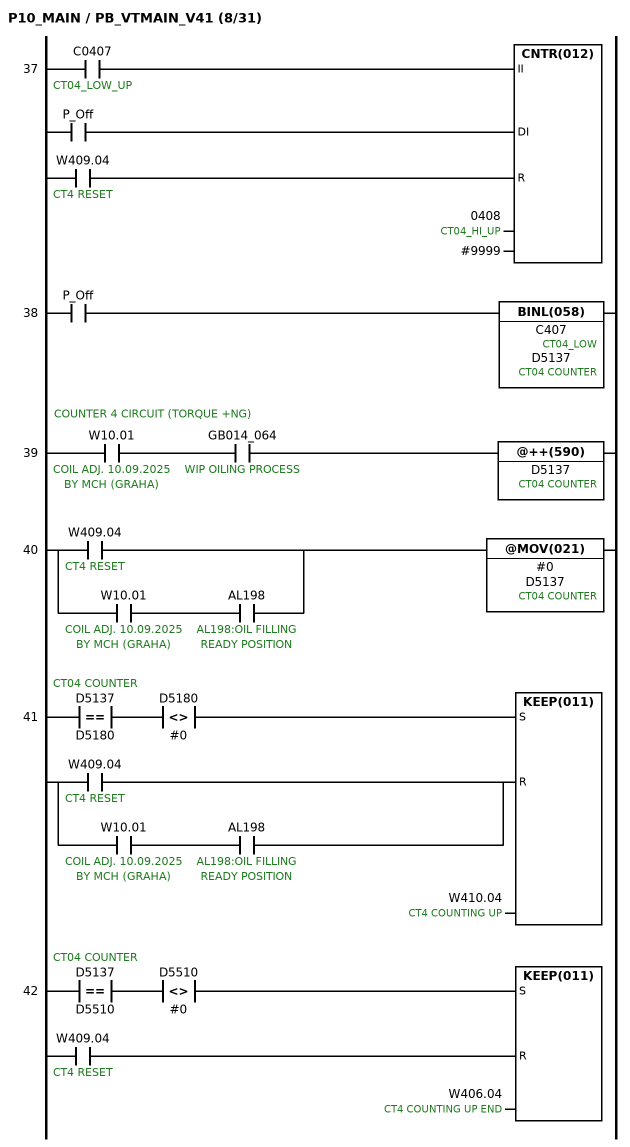
; [picture p96: P10_MAIN / PB_VTMAIN_V41, rungs 37-42]
; rung 37
LD C0407  ; CT04_LOW_UP
LD P_Off
LD W409.04  ; CT4 RESET
CNTR(012) 0408 #9999  ; CT04_HI_UP
; rung 38
LD P_Off
BINL(058) C407 D5137  ; CT04_LOW, CT04 COUNTER
; rung 39: COUNTER 4 CIRCUIT (TORQUE +NG)
LD W10.01  ; COIL ADJ. 10.09.2025 BY MCH (GRAHA)
AND GB014_064  ; WIP OILING PROCESS
@++(590) D5137  ; CT04 COUNTER
; rung 40
LD W409.04  ; CT4 RESET
LD W10.01  ; COIL ADJ. 10.09.2025 BY MCH (GRAHA)
AND AL198  ; AL198:OIL FILLING READY POSITION
ORLD
@MOV(021) #0 D5137  ; CT04 COUNTER
; rung 41
LD=L(301) D5137 D5180  ; CT04 COUNTER
AND<>L(306) D5180 #0
LD W409.04  ; CT4 RESET
LD W10.01  ; COIL ADJ. 10.09.2025 BY MCH (GRAHA)
AND AL198  ; AL198:OIL FILLING READY POSITION
ORLD
KEEP(011) W410.04  ; CT4 COUNTING UP
; rung 42
LD=L(301) D5137 D5510  ; CT04 COUNTER
AND<>L(306) D5510 #0
LD W409.04  ; CT4 RESET
KEEP(011) W406.04  ; CT4 COUNTING UP END

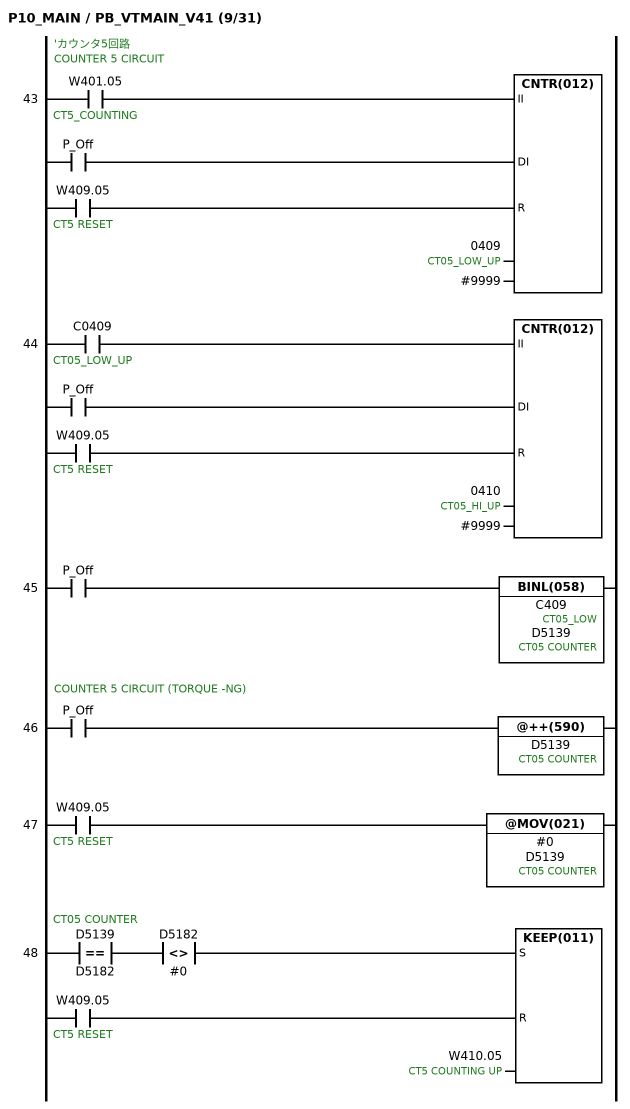
; rung 43: 'カウンタ5回路 / COUNTER 5 CIRCUIT
LD W401.05  ; CT5_COUNTING
LD P_Off
LD W409.05  ; CT5 RESET
CNTR(012) 0409 #9999  ; CT05_LOW_UP
; rung 44
LD C0409  ; CT05_LOW_UP
LD P_Off
LD W409.05  ; CT5 RESET
CNTR(012) 0410 #9999  ; CT05_HI_UP
; rung 45
LD P_Off
BINL(058) C409 D5139  ; CT05_LOW, CT05 COUNTER
; rung 46: COUNTER 5 CIRCUIT (TORQUE -NG)
LD P_Off
@++(590) D5139  ; CT05 COUNTER
; rung 47
LD W409.05  ; CT5 RESET
@MOV(021) #0 D5139  ; CT05 COUNTER
; rung 48
LD=L(301) D5139 D5182  ; CT05 COUNTER
AND<>L(306) D5182 #0
LD W409.05  ; CT5 RESET
KEEP(011) W410.05  ; CT5 COUNTING UP

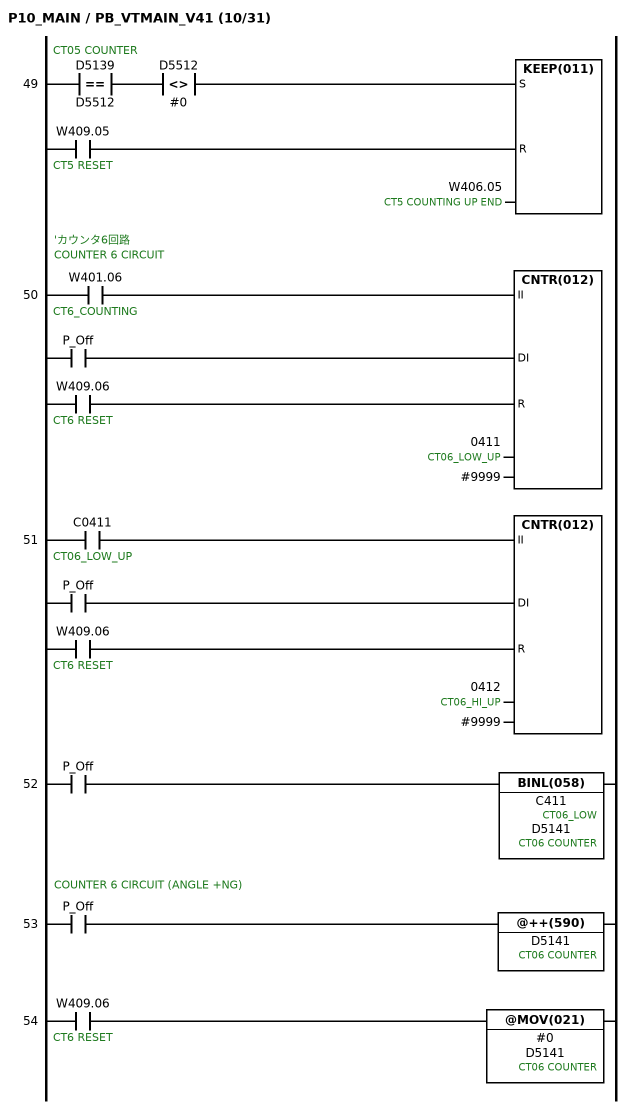
; rung 49
LD=L(301) D5139 D5512  ; CT05 COUNTER
AND<>L(306) D5512 #0
LD W409.05  ; CT5 RESET
KEEP(011) W406.05  ; CT5 COUNTING UP END
; rung 50: 'カウンタ6回路 / COUNTER 6 CIRCUIT
LD W401.06  ; CT6_COUNTING
LD P_Off
LD W409.06  ; CT6 RESET
CNTR(012) 0411 #9999  ; CT06_LOW_UP
; rung 51
LD C0411  ; CT06_LOW_UP
LD P_Off
LD W409.06  ; CT6 RESET
CNTR(012) 0412 #9999  ; CT06_HI_UP
; rung 52
LD P_Off
BINL(058) C411 D5141  ; CT06_LOW, CT06 COUNTER
; rung 53: COUNTER 6 CIRCUIT (ANGLE +NG)
LD P_Off
@++(590) D5141  ; CT06 COUNTER
; rung 54
LD W409.06  ; CT6 RESET
@MOV(021) #0 D5141  ; CT06 COUNTER

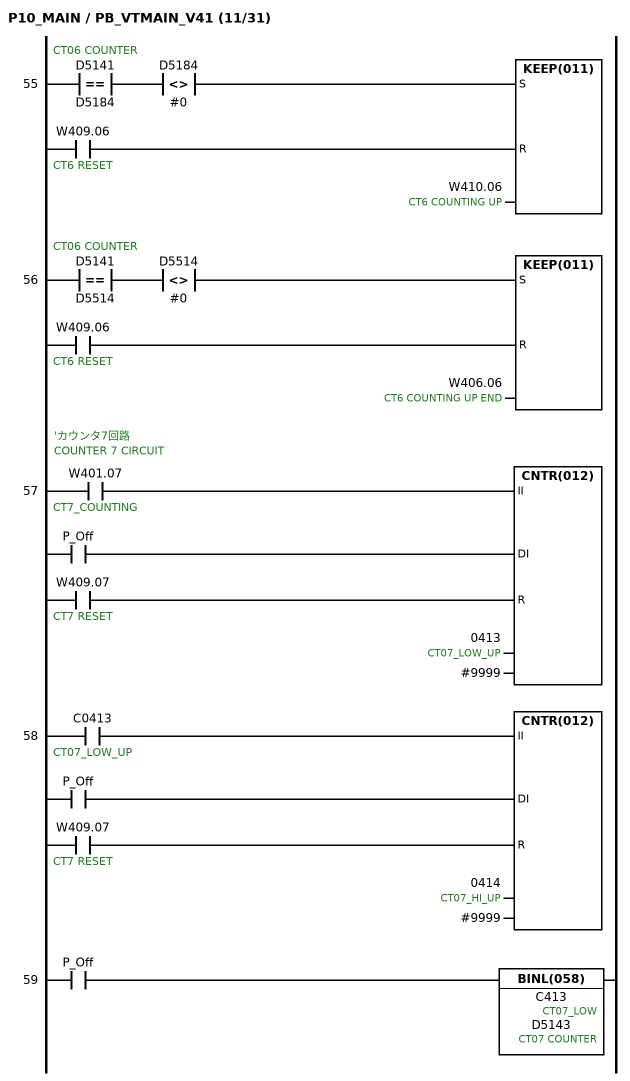
; rung 55
LD=L(301) D5141 D5184  ; CT06 COUNTER
AND<>L(306) D5184 #0
LD W409.06  ; CT6 RESET
KEEP(011) W410.06  ; CT6 COUNTING UP
; rung 56
LD=L(301) D5141 D5514  ; CT06 COUNTER
AND<>L(306) D5514 #0
LD W409.06  ; CT6 RESET
KEEP(011) W406.06  ; CT6 COUNTING UP END
; rung 57: 'カウンタ7回路 / COUNTER 7 CIRCUIT
LD W401.07  ; CT7_COUNTING
LD P_Off
LD W409.07  ; CT7 RESET
CNTR(012) 0413 #9999  ; CT07_LOW_UP
; rung 58
LD C0413  ; CT07_LOW_UP
LD P_Off
LD W409.07  ; CT7 RESET
CNTR(012) 0414 #9999  ; CT07_HI_UP
; rung 59
LD P_Off
BINL(058) C413 D5143  ; CT07_LOW, CT07 COUNTER

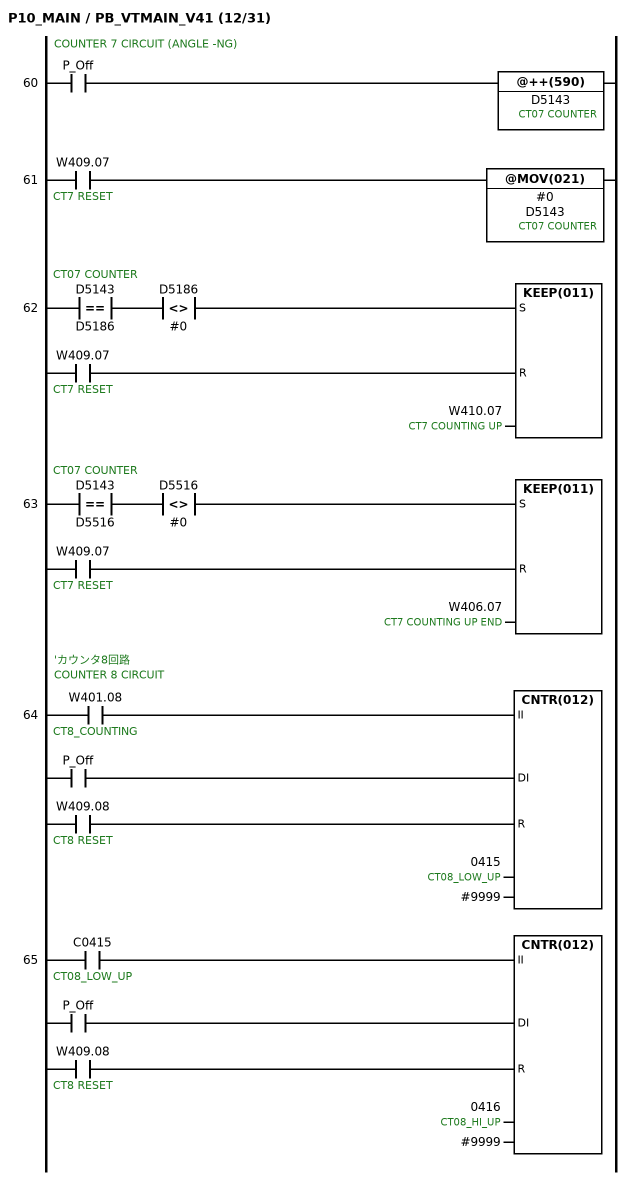
; rung 60: COUNTER 7 CIRCUIT (ANGLE -NG)
LD P_Off
@++(590) D5143  ; CT07 COUNTER
; rung 61
LD W409.07  ; CT7 RESET
@MOV(021) #0 D5143  ; CT07 COUNTER
; rung 62
LD=L(301) D5143 D5186  ; CT07 COUNTER
AND<>L(306) D5186 #0
LD W409.07  ; CT7 RESET
KEEP(011) W410.07  ; CT7 COUNTING UP
; rung 63
LD=L(301) D5143 D5516  ; CT07 COUNTER
AND<>L(306) D5516 #0
LD W409.07  ; CT7 RESET
KEEP(011) W406.07  ; CT7 COUNTING UP END
; rung 64: 'カウンタ8回路 / COUNTER 8 CIRCUIT
LD W401.08  ; CT8_COUNTING
LD P_Off
LD W409.08  ; CT8 RESET
CNTR(012) 0415 #9999  ; CT08_LOW_UP
; rung 65
LD C0415  ; CT08_LOW_UP
LD P_Off
LD W409.08  ; CT8 RESET
CNTR(012) 0416 #9999  ; CT08_HI_UP

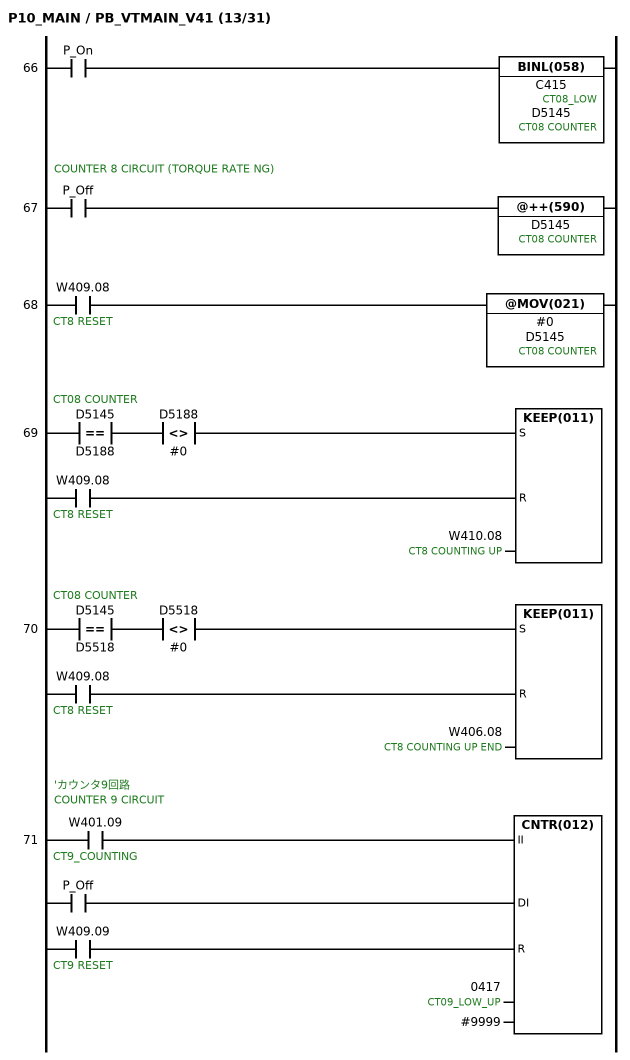
; rung 66
LD P_On
BINL(058) C415 D5145  ; CT08_LOW, CT08 COUNTER
; rung 67: COUNTER 8 CIRCUIT (TORQUE RATE NG)
LD P_Off
@++(590) D5145  ; CT08 COUNTER
; rung 68
LD W409.08  ; CT8 RESET
@MOV(021) #0 D5145  ; CT08 COUNTER
; rung 69
LD=L(301) D5145 D5188  ; CT08 COUNTER
AND<>L(306) D5188 #0
LD W409.08  ; CT8 RESET
KEEP(011) W410.08  ; CT8 COUNTING UP
; rung 70
LD=L(301) D5145 D5518  ; CT08 COUNTER
AND<>L(306) D5518 #0
LD W409.08  ; CT8 RESET
KEEP(011) W406.08  ; CT8 COUNTING UP END
; rung 71: 'カウンタ9回路 / COUNTER 9 CIRCUIT
LD W401.09  ; CT9_COUNTING
LD P_Off
LD W409.09  ; CT9 RESET
CNTR(012) 0417 #9999  ; CT09_LOW_UP

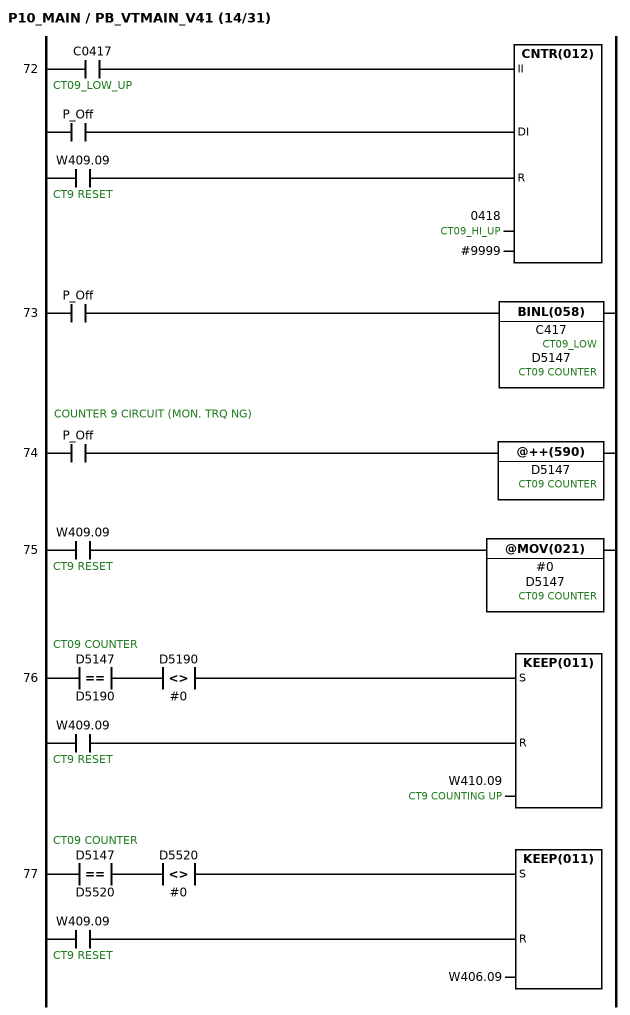
; rung 72
LD C0417  ; CT09_LOW_UP
LD P_Off
LD W409.09  ; CT9 RESET
CNTR(012) 0418 #9999  ; CT09_HI_UP
; rung 73
LD P_Off
BINL(058) C417 D5147  ; CT09_LOW, CT09 COUNTER
; rung 74: COUNTER 9 CIRCUIT (MON. TRQ NG)
LD P_Off
@++(590) D5147  ; CT09 COUNTER
; rung 75
LD W409.09  ; CT9 RESET
@MOV(021) #0 D5147  ; CT09 COUNTER
; rung 76
LD=L(301) D5147 D5190  ; CT09 COUNTER
AND<>L(306) D5190 #0
LD W409.09  ; CT9 RESET
KEEP(011) W410.09  ; CT9 COUNTING UP
; rung 77
LD=L(301) D5147 D5520  ; CT09 COUNTER
AND<>L(306) D5520 #0
LD W409.09  ; CT9 RESET
KEEP(011) W406.09

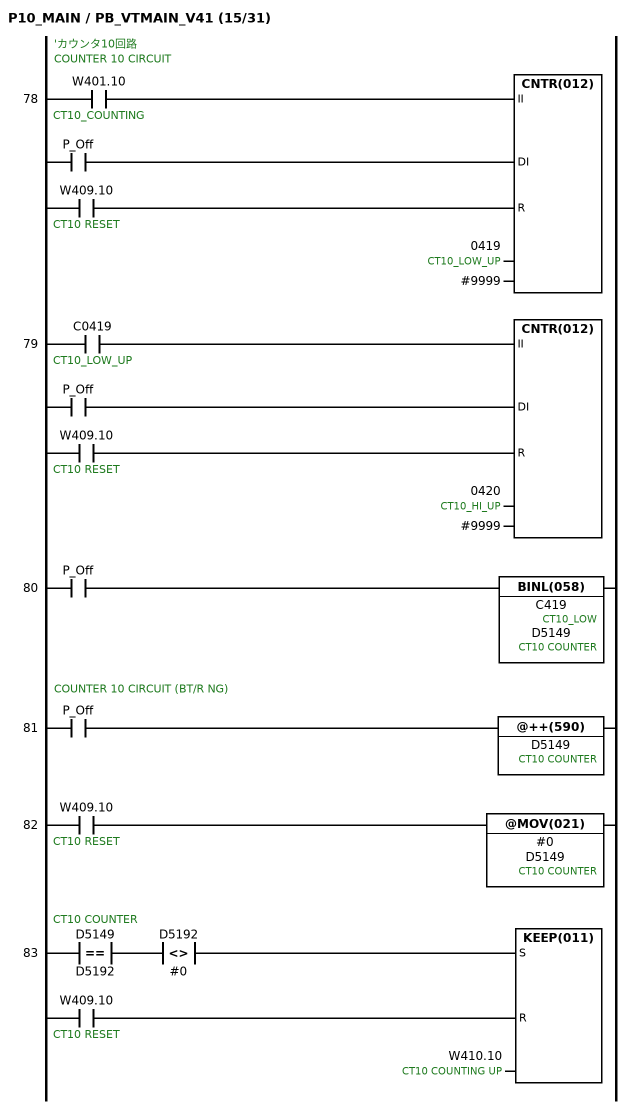
; rung 78: 'カウンタ10回路 / COUNTER 10 CIRCUIT
LD W401.10  ; CT10_COUNTING
LD P_Off
LD W409.10  ; CT10 RESET
CNTR(012) 0419 #9999  ; CT10_LOW_UP
; rung 79
LD C0419  ; CT10_LOW_UP
LD P_Off
LD W409.10  ; CT10 RESET
CNTR(012) 0420 #9999  ; CT10_HI_UP
; rung 80
LD P_Off
BINL(058) C419 D5149  ; CT10_LOW, CT10 COUNTER
; rung 81: COUNTER 10 CIRCUIT (BT/R NG)
LD P_Off
@++(590) D5149  ; CT10 COUNTER
; rung 82
LD W409.10  ; CT10 RESET
@MOV(021) #0 D5149  ; CT10 COUNTER
; rung 83
LD=L(301) D5149 D5192  ; CT10 COUNTER
AND<>L(306) D5192 #0
LD W409.10  ; CT10 RESET
KEEP(011) W410.10  ; CT10 COUNTING UP

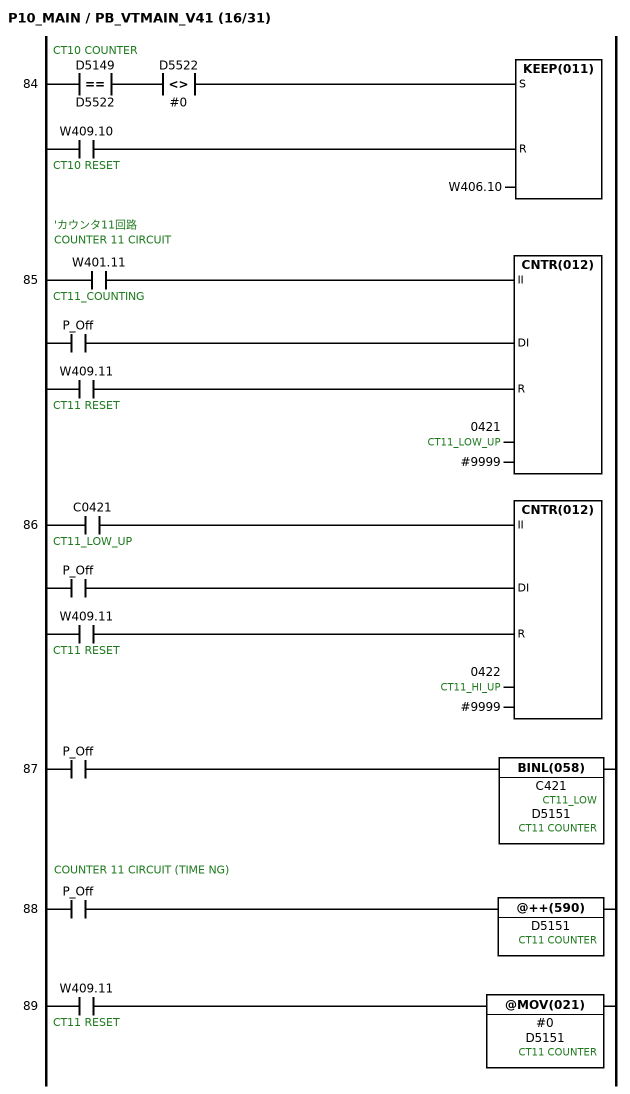
; rung 84
LD=L(301) D5149 D5522  ; CT10 COUNTER
AND<>L(306) D5522 #0
LD W409.10  ; CT10 RESET
KEEP(011) W406.10
; rung 85: 'カウンタ11回路 / COUNTER 11 CIRCUIT
LD W401.11  ; CT11_COUNTING
LD P_Off
LD W409.11  ; CT11 RESET
CNTR(012) 0421 #9999  ; CT11_LOW_UP
; rung 86
LD C0421  ; CT11_LOW_UP
LD P_Off
LD W409.11  ; CT11 RESET
CNTR(012) 0422 #9999  ; CT11_HI_UP
; rung 87
LD P_Off
BINL(058) C421 D5151  ; CT11_LOW, CT11 COUNTER
; rung 88: COUNTER 11 CIRCUIT (TIME NG)
LD P_Off
@++(590) D5151  ; CT11 COUNTER
; rung 89
LD W409.11  ; CT11 RESET
@MOV(021) #0 D5151  ; CT11 COUNTER

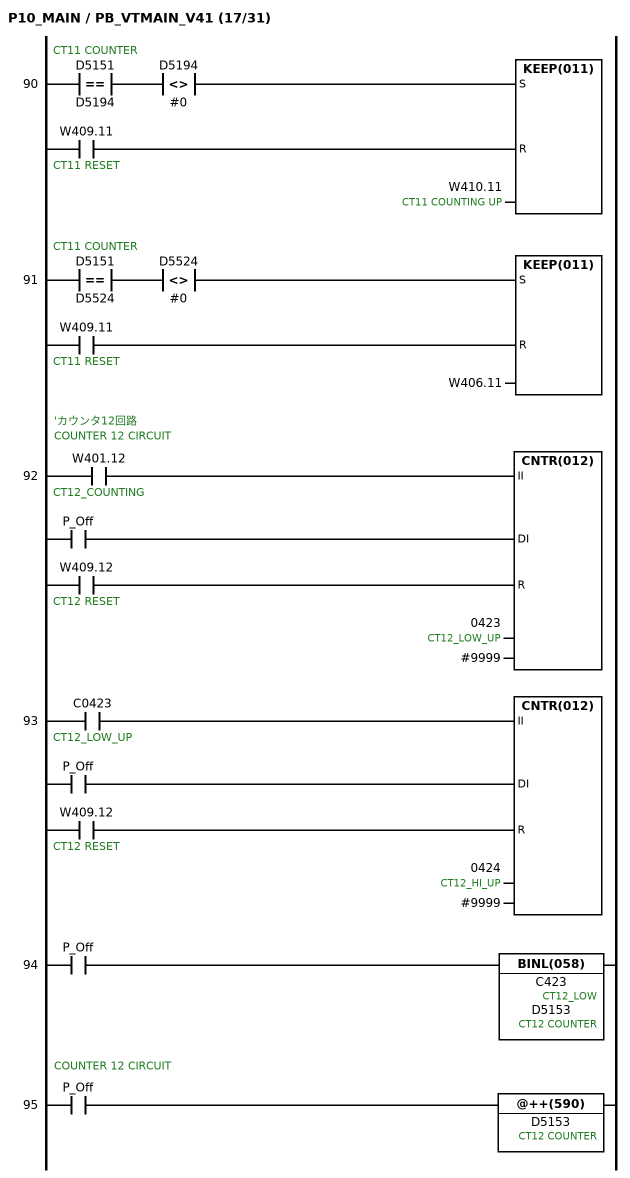
; rung 90
LD=L(301) D5151 D5194  ; CT11 COUNTER
AND<>L(306) D5194 #0
LD W409.11  ; CT11 RESET
KEEP(011) W410.11  ; CT11 COUNTING UP
; rung 91
LD=L(301) D5151 D5524  ; CT11 COUNTER
AND<>L(306) D5524 #0
LD W409.11  ; CT11 RESET
KEEP(011) W406.11
; rung 92: 'カウンタ12回路 / COUNTER 12 CIRCUIT
LD W401.12  ; CT12_COUNTING
LD P_Off
LD W409.12  ; CT12 RESET
CNTR(012) 0423 #9999  ; CT12_LOW_UP
; rung 93
LD C0423  ; CT12_LOW_UP
LD P_Off
LD W409.12  ; CT12 RESET
CNTR(012) 0424 #9999  ; CT12_HI_UP
; rung 94
LD P_Off
BINL(058) C423 D5153  ; CT12_LOW, CT12 COUNTER
; rung 95: COUNTER 12 CIRCUIT
LD P_Off
@++(590) D5153  ; CT12 COUNTER

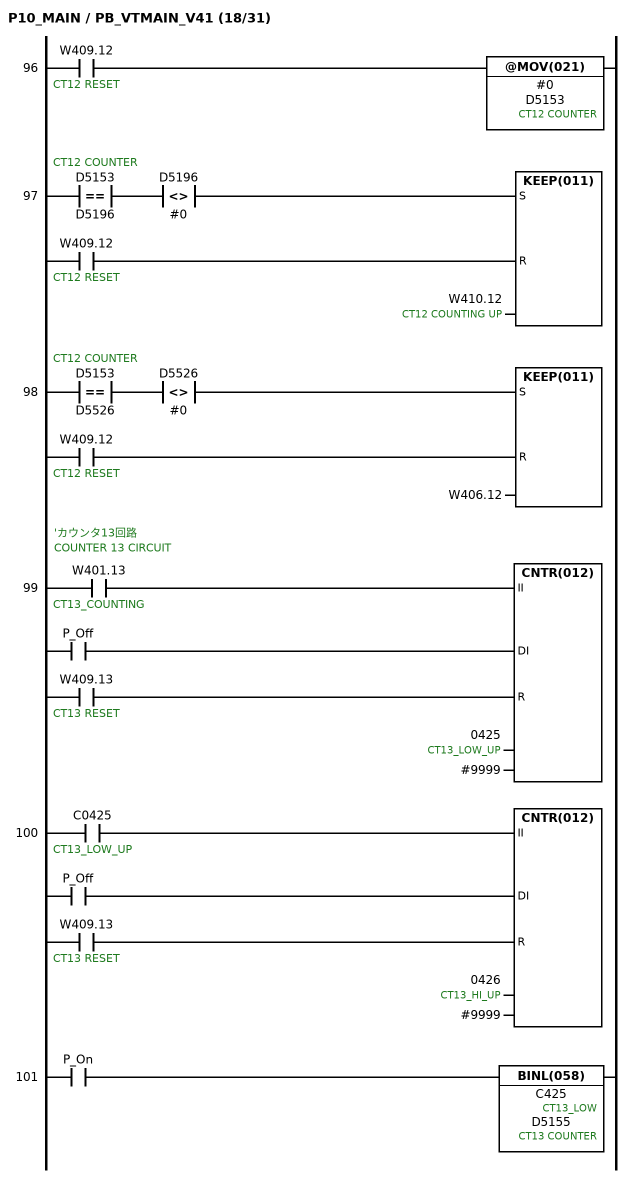
; rung 96
LD W409.12  ; CT12 RESET
@MOV(021) #0 D5153  ; CT12 COUNTER
; rung 97
LD=L(301) D5153 D5196  ; CT12 COUNTER
AND<>L(306) D5196 #0
LD W409.12  ; CT12 RESET
KEEP(011) W410.12  ; CT12 COUNTING UP
; rung 98
LD=L(301) D5153 D5526  ; CT12 COUNTER
AND<>L(306) D5526 #0
LD W409.12  ; CT12 RESET
KEEP(011) W406.12
; rung 99: 'カウンタ13回路 / COUNTER 13 CIRCUIT
LD W401.13  ; CT13_COUNTING
LD P_Off
LD W409.13  ; CT13 RESET
CNTR(012) 0425 #9999  ; CT13_LOW_UP
; rung 100
LD C0425  ; CT13_LOW_UP
LD P_Off
LD W409.13  ; CT13 RESET
CNTR(012) 0426 #9999  ; CT13_HI_UP
; rung 101
LD P_On
BINL(058) C425 D5155  ; CT13_LOW, CT13 COUNTER

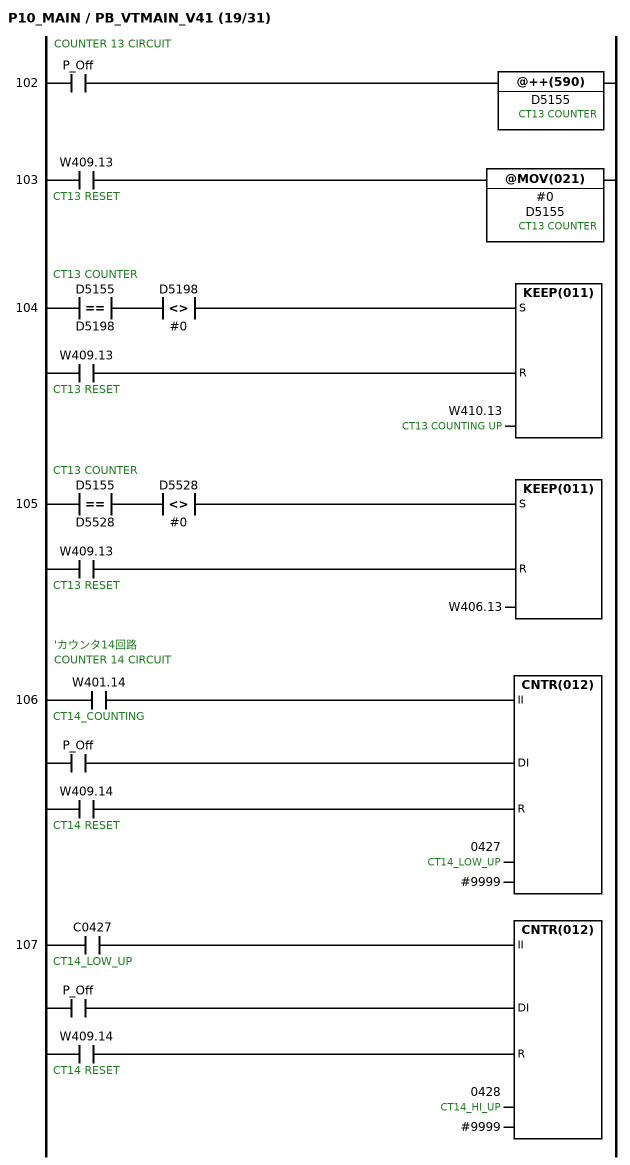
; rung 102: COUNTER 13 CIRCUIT
LD P_Off
@++(590) D5155  ; CT13 COUNTER
; rung 103
LD W409.13  ; CT13 RESET
@MOV(021) #0 D5155  ; CT13 COUNTER
; rung 104
LD=L(301) D5155 D5198  ; CT13 COUNTER
AND<>L(306) D5198 #0
LD W409.13  ; CT13 RESET
KEEP(011) W410.13  ; CT13 COUNTING UP
; rung 105
LD=L(301) D5155 D5528  ; CT13 COUNTER
AND<>L(306) D5528 #0
LD W409.13  ; CT13 RESET
KEEP(011) W406.13
; rung 106: 'カウンタ14回路 / COUNTER 14 CIRCUIT
LD W401.14  ; CT14_COUNTING
LD P_Off
LD W409.14  ; CT14 RESET
CNTR(012) 0427 #9999  ; CT14_LOW_UP
; rung 107
LD C0427  ; CT14_LOW_UP
LD P_Off
LD W409.14  ; CT14 RESET
CNTR(012) 0428 #9999  ; CT14_HI_UP

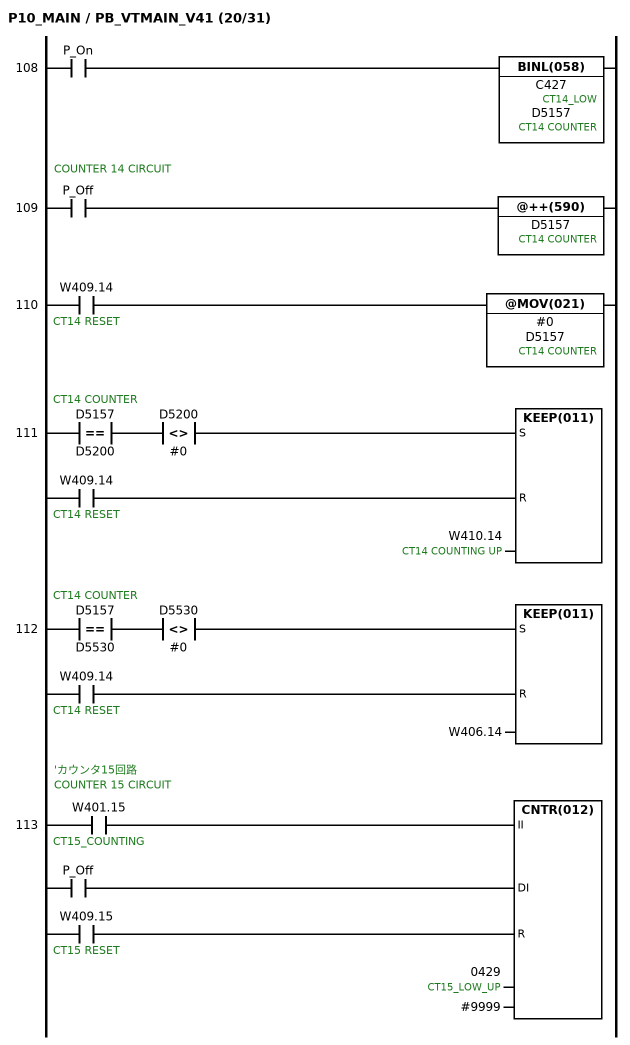
; rung 108
LD P_On
BINL(058) C427 D5157  ; CT14_LOW, CT14 COUNTER
; rung 109: COUNTER 14 CIRCUIT
LD P_Off
@++(590) D5157  ; CT14 COUNTER
; rung 110
LD W409.14  ; CT14 RESET
@MOV(021) #0 D5157  ; CT14 COUNTER
; rung 111
LD=L(301) D5157 D5200  ; CT14 COUNTER
AND<>L(306) D5200 #0
LD W409.14  ; CT14 RESET
KEEP(011) W410.14  ; CT14 COUNTING UP
; rung 112
LD=L(301) D5157 D5530  ; CT14 COUNTER
AND<>L(306) D5530 #0
LD W409.14  ; CT14 RESET
KEEP(011) W406.14
; rung 113: 'カウンタ15回路 / COUNTER 15 CIRCUIT
LD W401.15  ; CT15_COUNTING
LD P_Off
LD W409.15  ; CT15 RESET
CNTR(012) 0429 #9999  ; CT15_LOW_UP

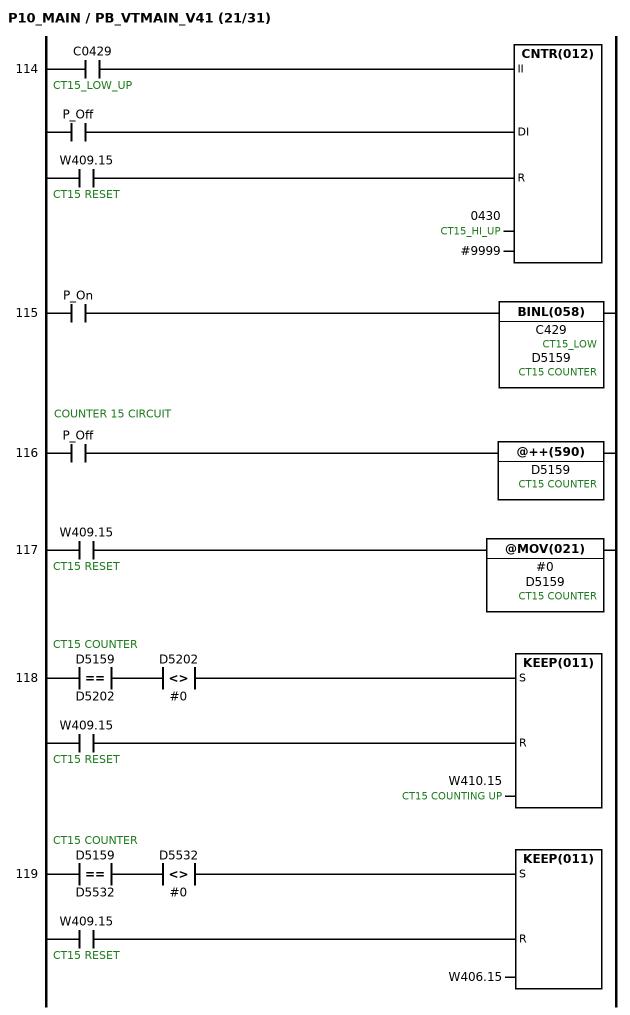
; rung 114
LD C0429  ; CT15_LOW_UP
LD P_Off
LD W409.15  ; CT15 RESET
CNTR(012) 0430 #9999  ; CT15_HI_UP
; rung 115
LD P_On
BINL(058) C429 D5159  ; CT15_LOW, CT15 COUNTER
; rung 116: COUNTER 15 CIRCUIT
LD P_Off
@++(590) D5159  ; CT15 COUNTER
; rung 117
LD W409.15  ; CT15 RESET
@MOV(021) #0 D5159  ; CT15 COUNTER
; rung 118
LD=L(301) D5159 D5202  ; CT15 COUNTER
AND<>L(306) D5202 #0
LD W409.15  ; CT15 RESET
KEEP(011) W410.15  ; CT15 COUNTING UP
; rung 119
LD=L(301) D5159 D5532  ; CT15 COUNTER
AND<>L(306) D5532 #0
LD W409.15  ; CT15 RESET
KEEP(011) W406.15

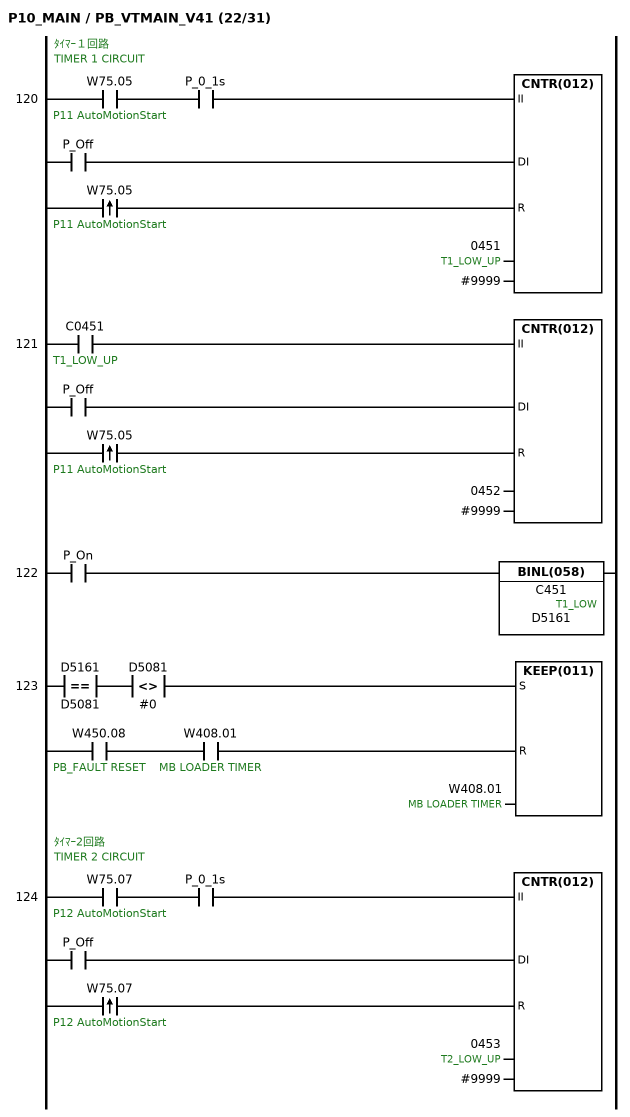
; rung 120: ﾀｲﾏｰ１回路 / TIMER 1 CIRCUIT
LD W75.05  ; P11 AutoMotionStart
AND P_0_1s
LD P_Off
@LD W75.05  ; P11 AutoMotionStart
CNTR(012) 0451 #9999  ; T1_LOW_UP
; rung 121
LD C0451  ; T1_LOW_UP
LD P_Off
@LD W75.05  ; P11 AutoMotionStart
CNTR(012) 0452 #9999
; rung 122
LD P_On
BINL(058) C451 D5161  ; T1_LOW
; rung 123
LD=(300) D5161 D5081
AND<>(305) D5081 #0
LD W450.08  ; PB_FAULT RESET
AND W408.01  ; MB LOADER TIMER
KEEP(011) W408.01  ; MB LOADER TIMER
; rung 124: ﾀｲﾏｰ2回路 / TIMER 2 CIRCUIT
LD W75.07  ; P12 AutoMotionStart
AND P_0_1s
LD P_Off
@LD W75.07  ; P12 AutoMotionStart
CNTR(012) 0453 #9999  ; T2_LOW_UP

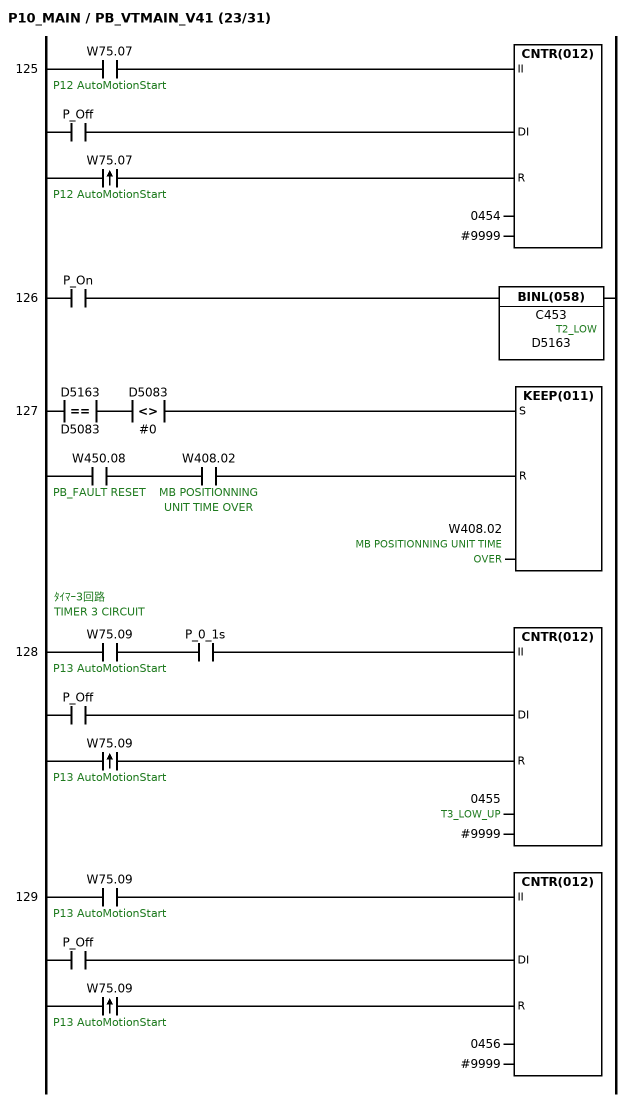
; rung 125
LD W75.07  ; P12 AutoMotionStart
LD P_Off
@LD W75.07  ; P12 AutoMotionStart
CNTR(012) 0454 #9999
; rung 126
LD P_On
BINL(058) C453 D5163  ; T2_LOW
; rung 127
LD=(300) D5163 D5083
AND<>(305) D5083 #0
LD W450.08  ; PB_FAULT RESET
AND W408.02  ; MB POSITIONNING UNIT TIME OVER
KEEP(011) W408.02  ; MB POSITIONNING UNIT TIME OVER
; rung 128: ﾀｲﾏｰ3回路 / TIMER 3 CIRCUIT
LD W75.09  ; P13 AutoMotionStart
AND P_0_1s
LD P_Off
@LD W75.09  ; P13 AutoMotionStart
CNTR(012) 0455 #9999  ; T3_LOW_UP
; rung 129
LD W75.09  ; P13 AutoMotionStart
LD P_Off
@LD W75.09  ; P13 AutoMotionStart
CNTR(012) 0456 #9999

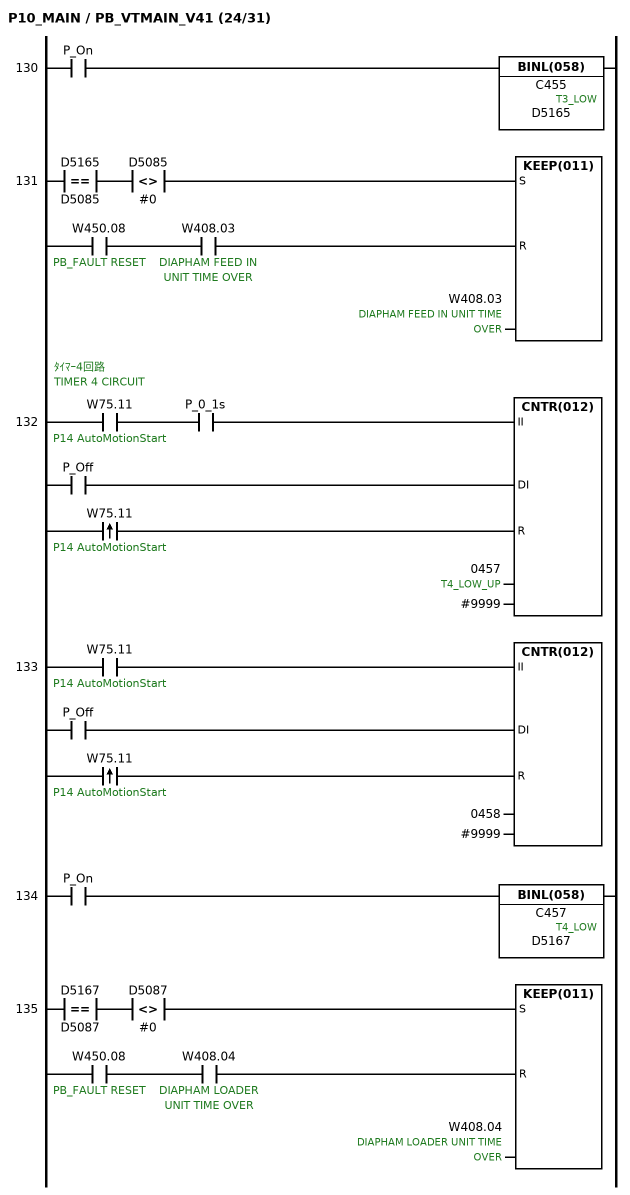
; rung 130
LD P_On
BINL(058) C455 D5165  ; T3_LOW
; rung 131
LD=(300) D5165 D5085
AND<>(305) D5085 #0
LD W450.08  ; PB_FAULT RESET
AND W408.03  ; DIAPHAM FEED IN UNIT TIME OVER
KEEP(011) W408.03  ; DIAPHAM FEED IN UNIT TIME OVER
; rung 132: ﾀｲﾏｰ4回路 / TIMER 4 CIRCUIT
LD W75.11  ; P14 AutoMotionStart
AND P_0_1s
LD P_Off
@LD W75.11  ; P14 AutoMotionStart
CNTR(012) 0457 #9999  ; T4_LOW_UP
; rung 133
LD W75.11  ; P14 AutoMotionStart
LD P_Off
@LD W75.11  ; P14 AutoMotionStart
CNTR(012) 0458 #9999
; rung 134
LD P_On
BINL(058) C457 D5167  ; T4_LOW
; rung 135
LD=(300) D5167 D5087
AND<>(305) D5087 #0
LD W450.08  ; PB_FAULT RESET
AND W408.04  ; DIAPHAM LOADER UNIT TIME OVER
KEEP(011) W408.04  ; DIAPHAM LOADER UNIT TIME OVER

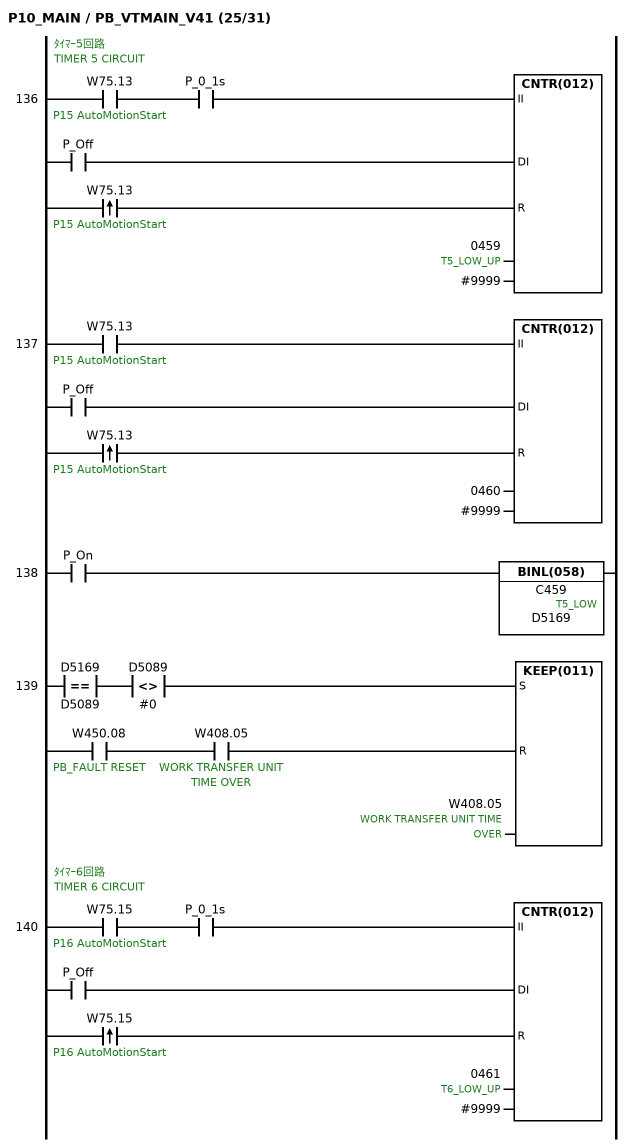
; rung 136: ﾀｲﾏｰ5回路 / TIMER 5 CIRCUIT
LD W75.13  ; P15 AutoMotionStart
AND P_0_1s
LD P_Off
@LD W75.13  ; P15 AutoMotionStart
CNTR(012) 0459 #9999  ; T5_LOW_UP
; rung 137
LD W75.13  ; P15 AutoMotionStart
LD P_Off
@LD W75.13  ; P15 AutoMotionStart
CNTR(012) 0460 #9999
; rung 138
LD P_On
BINL(058) C459 D5169  ; T5_LOW
; rung 139
LD=(300) D5169 D5089
AND<>(305) D5089 #0
LD W450.08  ; PB_FAULT RESET
AND W408.05  ; WORK TRANSFER UNIT TIME OVER
KEEP(011) W408.05  ; WORK TRANSFER UNIT TIME OVER
; rung 140: ﾀｲﾏｰ6回路 / TIMER 6 CIRCUIT
LD W75.15  ; P16 AutoMotionStart
AND P_0_1s
LD P_Off
@LD W75.15  ; P16 AutoMotionStart
CNTR(012) 0461 #9999  ; T6_LOW_UP

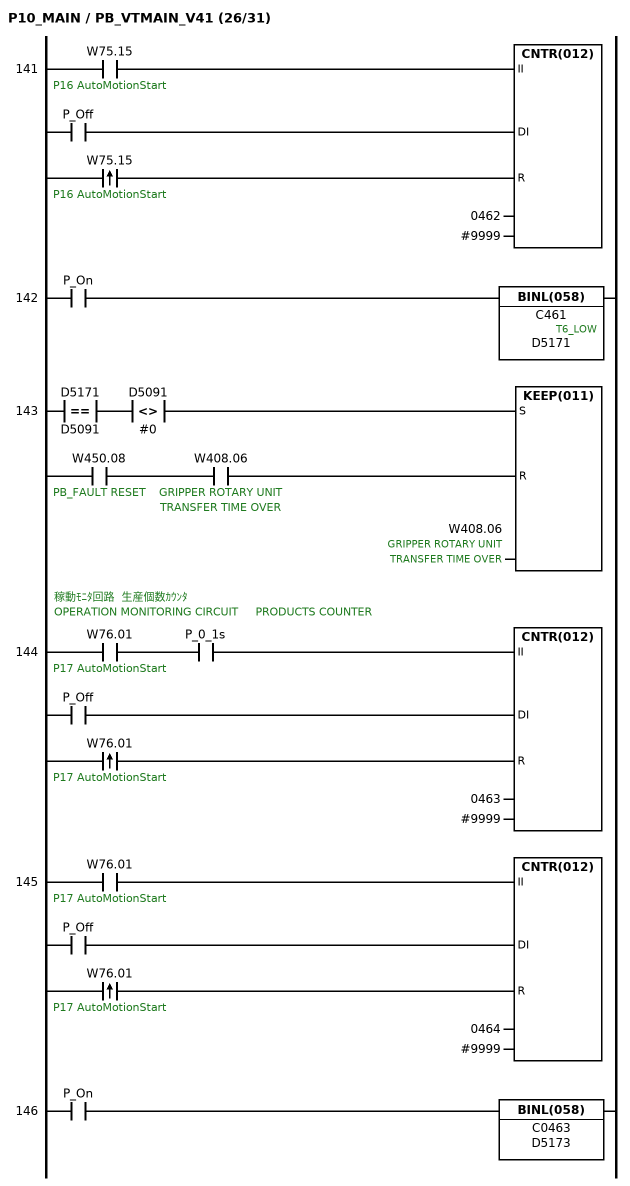
; rung 141
LD W75.15  ; P16 AutoMotionStart
LD P_Off
@LD W75.15  ; P16 AutoMotionStart
CNTR(012) 0462 #9999
; rung 142
LD P_On
BINL(058) C461 D5171  ; T6_LOW
; rung 143
LD=(300) D5171 D5091
AND<>(305) D5091 #0
LD W450.08  ; PB_FAULT RESET
AND W408.06  ; GRIPPER ROTARY UNIT TRANSFER TIME OVER
KEEP(011) W408.06  ; GRIPPER ROTARY UNIT TRANSFER TIME OVER
; rung 144: 稼動ﾓﾆﾀ回路  生産個数ｶｳﾝﾀ / OPERATION MONITORING CIRCUIT     PRODUCTS COUNTER
LD W76.01  ; P17 AutoMotionStart
AND P_0_1s
LD P_Off
@LD W76.01  ; P17 AutoMotionStart
CNTR(012) 0463 #9999
; rung 145
LD W76.01  ; P17 AutoMotionStart
LD P_Off
@LD W76.01  ; P17 AutoMotionStart
CNTR(012) 0464 #9999
; rung 146
LD P_On
BINL(058) C0463 D5173

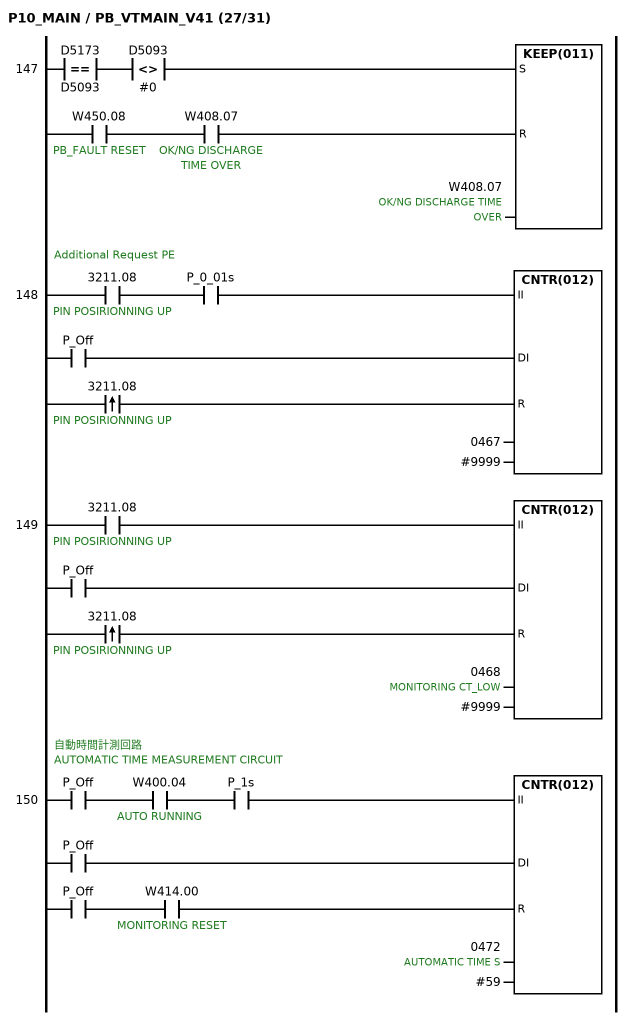
; rung 147
LD=(300) D5173 D5093
AND<>(305) D5093 #0
LD W450.08  ; PB_FAULT RESET
AND W408.07  ; OK/NG DISCHARGE TIME OVER
KEEP(011) W408.07  ; OK/NG DISCHARGE TIME OVER
; rung 148: Additional Request PE
LD 3211.08  ; PIN POSIRIONNING UP
AND P_0_01s
LD P_Off
@LD 3211.08  ; PIN POSIRIONNING UP
CNTR(012) 0467 #9999
; rung 149
LD 3211.08  ; PIN POSIRIONNING UP
LD P_Off
@LD 3211.08  ; PIN POSIRIONNING UP
CNTR(012) 0468 #9999  ; MONITORING CT_LOW
; rung 150: 自動時間計測回路 / AUTOMATIC TIME MEASUREMENT CIRCUIT
LD P_Off
AND W400.04  ; AUTO RUNNING
AND P_1s
LD P_Off
LD P_Off
AND W414.00  ; MONITORING RESET
CNTR(012) 0472 #59  ; AUTOMATIC TIME S

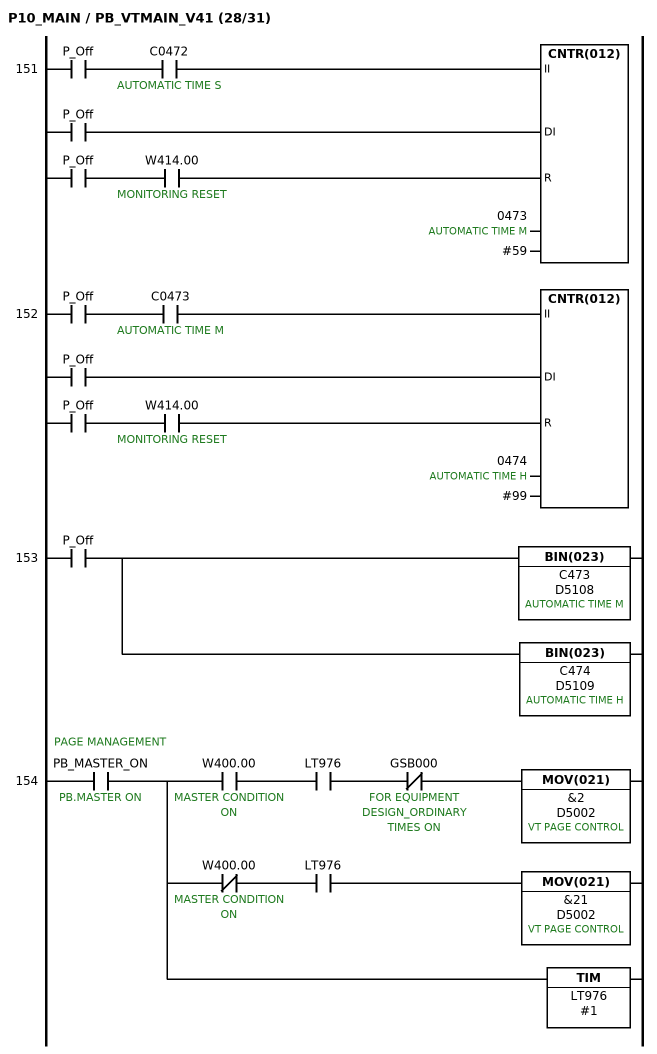
; rung 151
LD P_Off
AND C0472  ; AUTOMATIC TIME S
LD P_Off
LD P_Off
AND W414.00  ; MONITORING RESET
CNTR(012) 0473 #59  ; AUTOMATIC TIME M
; rung 152
LD P_Off
AND C0473  ; AUTOMATIC TIME M
LD P_Off
LD P_Off
AND W414.00  ; MONITORING RESET
CNTR(012) 0474 #99  ; AUTOMATIC TIME H
; rung 153
LD P_Off
BIN(023) C473 D5108  ; AUTOMATIC TIME M
BIN(023) C474 D5109  ; AUTOMATIC TIME H
; rung 154: PAGE MANAGEMENT
LD PB_MASTER_ON  ; PB.MASTER ON
OUT TR0
AND W400.00  ; MASTER CONDITION ON
AND LT976
ANDNOT GSB000  ; FOR EQUIPMENT DESIGN_ORDINARY TIMES ON
MOV(021) &2 D5002  ; VT PAGE CONTROL
LD TR0
ANDNOT W400.00  ; MASTER CONDITION ON
AND LT976
MOV(021) &21 D5002  ; VT PAGE CONTROL
LD TR0
TIM LT976 #1

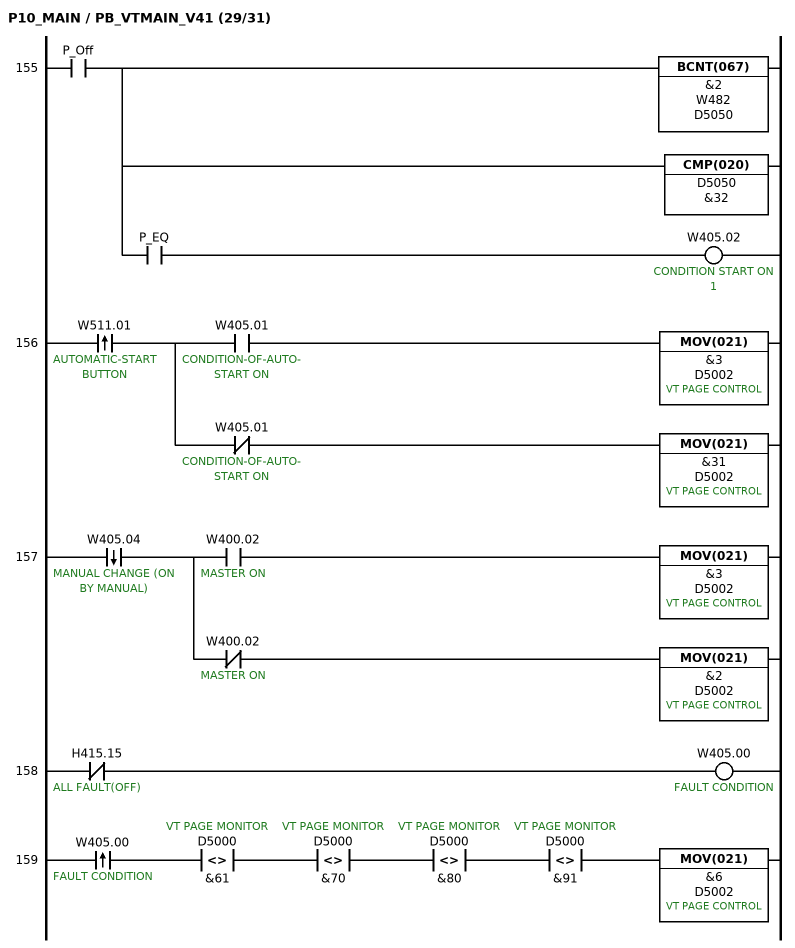
; rung 155
LD P_Off
BCNT(067) &2 W482 D5050
CMP(020) D5050 &32
AND P_EQ
OUT W405.02  ; CONDITION START ON 1
; rung 156
@LD W511.01  ; AUTOMATIC-START BUTTON
OUT TR0
AND W405.01  ; CONDITION-OF-AUTO-START ON
MOV(021) &3 D5002  ; VT PAGE CONTROL
LD TR0
ANDNOT W405.01  ; CONDITION-OF-AUTO-START ON
MOV(021) &31 D5002  ; VT PAGE CONTROL
; rung 157
%LD W405.04  ; MANUAL CHANGE (ON BY MANUAL)
OUT TR0
AND W400.02  ; MASTER ON
MOV(021) &3 D5002  ; VT PAGE CONTROL
LD TR0
ANDNOT W400.02  ; MASTER ON
MOV(021) &2 D5002  ; VT PAGE CONTROL
; rung 158
LDNOT H415.15  ; ALL FAULT(OFF)
OUT W405.00  ; FAULT CONDITION
; rung 159
@LD W405.00  ; FAULT CONDITION
AND<>(305) D5000 &61  ; VT PAGE MONITOR
AND<>(305) D5000 &70  ; VT PAGE MONITOR
AND<>(305) D5000 &80  ; VT PAGE MONITOR
AND<>(305) D5000 &91  ; VT PAGE MONITOR
MOV(021) &6 D5002  ; VT PAGE CONTROL

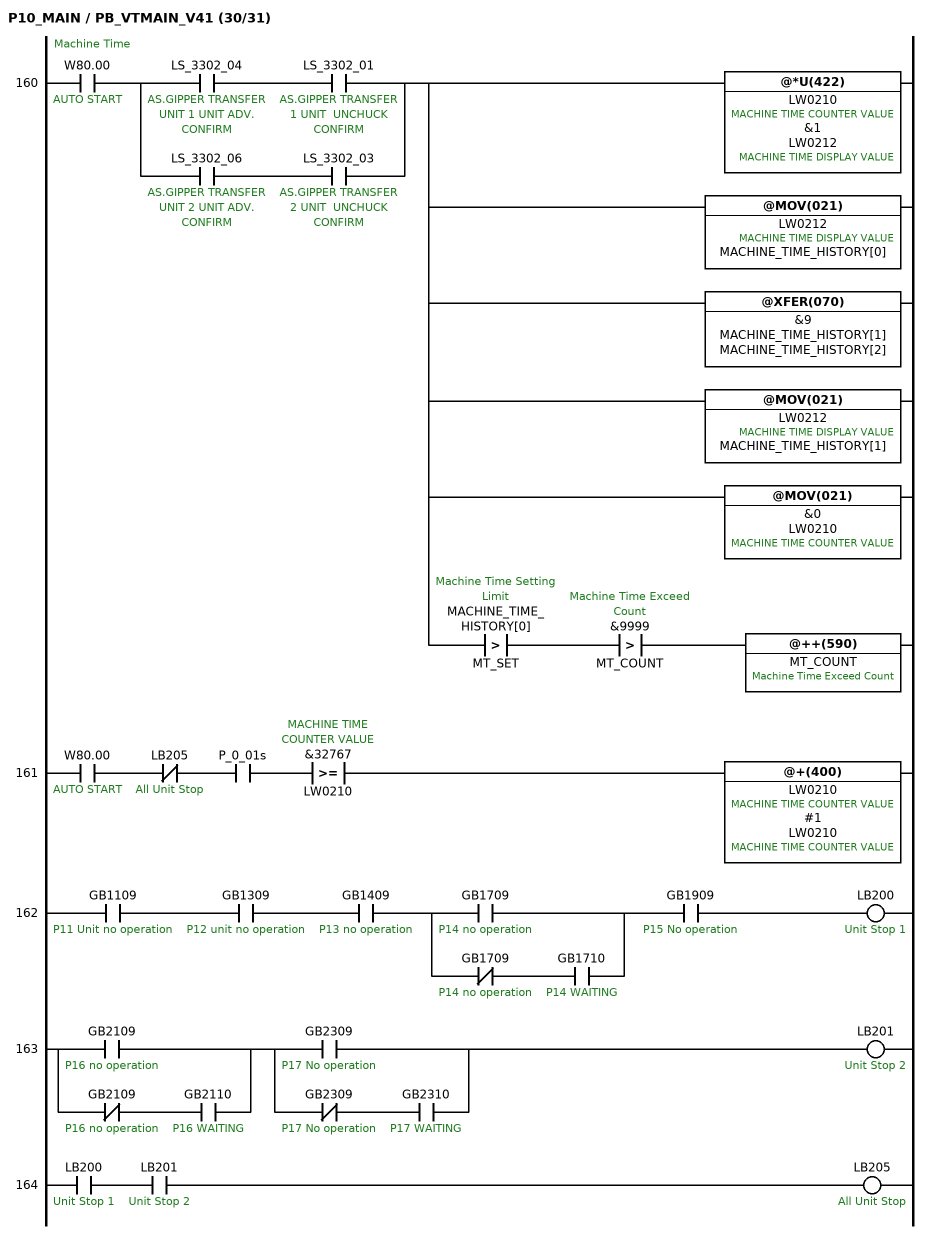
; rung 160: Machine Time
LD W80.00  ; AUTO START
LD LS_3302_04  ; AS.GIPPER TRANSFER UNIT 1 UNIT ADV. CONFIRM
AND LS_3302_01  ; AS.GIPPER TRANSFER 1 UNIT  UNCHUCK CONFIRM
LD LS_3302_06  ; AS.GIPPER TRANSFER UNIT 2 UNIT ADV. CONFIRM
AND LS_3302_03  ; AS.GIPPER TRANSFER 2 UNIT  UNCHUCK CONFIRM
ORLD
ANDLD
@*U(422) LW0210 &1 LW0212  ; MACHINE TIME COUNTER VALUE, MACHINE TIME DISPLAY VALUE
@MOV(021) LW0212 MACHINE_TIME_HISTORY[0]  ; MACHINE TIME DISPLAY VALUE
@XFER(070) &9 MACHINE_TIME_HISTORY[1] MACHINE_TIME_HISTORY[2]
@MOV(021) LW0212 MACHINE_TIME_HISTORY[1]  ; MACHINE TIME DISPLAY VALUE
@MOV(021) &0 LW0210  ; MACHINE TIME COUNTER VALUE
AND>(320) MACHINE_TIME_HISTORY[0] MT_SET  ; Machine Time Setting Limit
AND>(320) &9999 MT_COUNT  ; Machine Time Exceed Count
@++(590) MT_COUNT  ; Machine Time Exceed Count
; rung 161
LD W80.00  ; AUTO START
ANDNOT LB205  ; All Unit Stop
AND P_0_01s
AND>=(325) &32767 LW0210  ; MACHINE TIME COUNTER VALUE
@+(400) LW0210 #1 LW0210  ; MACHINE TIME COUNTER VALUE
; rung 162
LD GB1109  ; P11 Unit no operation
AND GB1309  ; P12 unit no operation
AND GB1409  ; P13 no operation
LD GB1709  ; P14 no operation
LDNOT GB1709  ; P14 no operation
AND GB1710  ; P14 WAITING
ORLD
ANDLD
AND GB1909  ; P15 No operation
OUT LB200  ; Unit Stop 1
; rung 163
LD GB2109  ; P16 no operation
LDNOT GB2109  ; P16 no operation
AND GB2110  ; P16 WAITING
ORLD
LD GB2309  ; P17 No operation
LDNOT GB2309  ; P17 No operation
AND GB2310  ; P17 WAITING
ORLD
ANDLD
OUT LB201  ; Unit Stop 2
; rung 164
LD LB200  ; Unit Stop 1
AND LB201  ; Unit Stop 2
OUT LB205  ; All Unit Stop

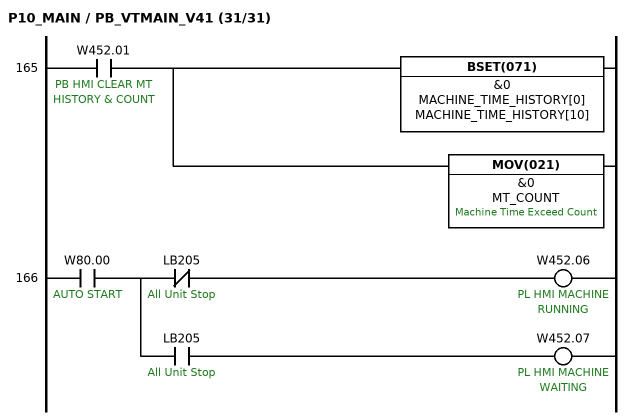
; rung 165
LD W452.01  ; PB HMI CLEAR MT HISTORY & COUNT
BSET(071) &0 MACHINE_TIME_HISTORY[0] MACHINE_TIME_HISTORY[10]
MOV(021) &0 MT_COUNT  ; Machine Time Exceed Count
; rung 166
LD W80.00  ; AUTO START
OUT TR0
ANDNOT LB205  ; All Unit Stop
OUT W452.06  ; PL HMI MACHINE RUNNING
LD TR0
AND LB205  ; All Unit Stop
OUT W452.07  ; PL HMI MACHINE WAITING

### Section END
; rung 0
END(001)

## Program P11_MB_LOADER (cyclic task 1)
Local symbols
GB011_004 E0_6.05 BOOL  ; Slide fwd Request
GB016_005 E0_6.06 BOOL  ; Forward allowed
GB1101 E0_6.07 BOOL  ; P11 Unit NO operation
LB100 E0_6.08 BOOL  ; P11 CycleStart
LB1000 E0_6.09 BOOL  ; AUTO START BEGIN
LB1000_1 E0_6.10 BOOL  ; Loader 1Check
LB1000_2 E0_6.11 BOOL  ; Have work
LB1000_3 E0_6.12 BOOL  ; Not have work
LB1001 E0_6.13 BOOL  ; MB LoadIn  DOWN
LB1002 E0_6.14 BOOL  ; MB LoadIn DOWN CONF
LB1003 E0_6.15 BOOL  ; MAGNETIZE 1 START
LB1004 E0_7.00 BOOL  ; MAGNETIZE 1 CONF
LB1005 E0_7.01 BOOL  ; LB LoadIn UP
LB1006 E0_7.02 BOOL  ; LB LoadIn UP CONF
LB1007 E0_7.03 BOOL  ; M&B LOAD UNIT SLIDE ADV.
LB1008 E0_7.04 BOOL  ; M&B LOAD UNIT SLIDE ADV.CONF
LB1009 E0_7.05 BOOL  ; M&B LOAD IN DOWN
LB101 E0_7.06 BOOL  ; Takeout Positioning
LB1010 E0_7.07 BOOL  ; M&B LOAD IN DOWN CONF
LB1011 E0_7.08 BOOL  ; M&B LOAD IN DEMAGNETIZW START
LB1012 E0_7.09 BOOL  ; M&B LOAD IN DEMAGNETIZW START CONF
LB1013 E0_7.10 BOOL  ; M&B LOAD IN UP
LB1014 E0_7.11 BOOL  ; M&B LOAD IN UP CONF
LB1015 E0_7.12 BOOL  ; AUTO START BEGIN
LB1015_1 E0_7.13 BOOL  ; Loader 1 check
LB1015_2 E0_7.14 BOOL  ; Have work
LB1015_3 E0_7.15 BOOL  ; Not have work
LB1016 E0_8.00 BOOL  ; MB LoadIn  DOWN
LB1017 E0_8.01 BOOL  ; MB LoadIn  DOWN CONF
LB1018 E0_8.02 BOOL  ; MB LoadOut  DOWN
LB1019 E0_8.03 BOOL  ; MB LoadOut DOWN CONF
LB102 E0_8.04 BOOL  ; Takeout Vacuum  & Positioning
LB1020 E0_8.05 BOOL  ; MB LoadOut UNIT DOWN
LB1021 E0_8.06 BOOL  ; MB LoadOut UNIT DOWN CONF
LB1022 E0_8.07 BOOL  ; MAGNETIZE 1 START
LB1023 E0_8.08 BOOL  ; MAGNETIZE 1 CONF
LB1024 E0_8.09 BOOL  ; MAGNETIZE 2 START
LB1025 E0_8.10 BOOL  ; MAGNETIZE 2 CONF
LB1026 E0_8.11 BOOL  ; LB LoadIn UP
LB1027 E0_8.12 BOOL  ; LB LoadIn UP CONF
LB1028 E0_8.13 BOOL  ; MB LoadOut  UP
LB1029 E0_8.14 BOOL  ; MB LoadOut  UP CONF
LB103 E0_8.15 BOOL  ; Takeout Vacuum
LB1030 E0_9.00 BOOL  ; MB LoadOut UNIT UP
LB1031 E0_9.01 BOOL  ; MB LoadOut UNIT UP CONF
LB1032 E0_9.02 BOOL  ; M&B LOAD UNIT SLIDE ADV.
LB1033 E0_9.03 BOOL  ; M&B LOAD UNIT SLIDE ADV. CONF
LB1034 E0_9.04 BOOL  ; M&B LOAD IN DOWN
LB1035 E0_9.05 BOOL  ; M&B LOAD IN DOWN CONF
LB1036 E0_9.06 BOOL  ; MB LoadOut  DOWN
LB1037 E0_9.07 BOOL  ; MB LoadOut Unit  DOWN
LB1038 E0_9.08 BOOL  ; MB LoadOut  DOWN CONF
LB1039 E0_9.09 BOOL  ; MB LoadOut UNIT DOWN CONF
LB104 E0_9.10 BOOL  ; Take in Vacuum
LB1040 E0_9.11 BOOL  ; M&B LOAD IN DEMAGNETIZW START
LB1041 E0_9.12 BOOL  ; M&B LOAD IN DEMAGNETIZW START CONF
LB1042 E0_9.13 BOOL  ; M&B LOAD OUT DEMAGNETIZW START
LB1043 E0_9.14 BOOL  ; M&B LOAD OUT DEMAGNETIZW START CONF
LB1044 E0_9.15 BOOL  ; M&B LOAD IN UP
LB1045 E0_10.00 BOOL  ; M&B LOAD IN UP CONF
LB1046 E0_10.01 BOOL  ; MB LoadOut  UP
LB1047 E0_10.02 BOOL  ; MB LoadOut  UP CONF
LB1048 E0_10.03 BOOL  ; MB LoadOut  UP CONF
LB1049 E0_10.04 BOOL  ; MB LoadOut UNIT UP CONF
LB105 E0_10.05 BOOL  ; Take in Positioning & Slide
LB1050 E0_10.06 BOOL  ; AUTO START BEGIN
LB1051 E0_10.07 BOOL  ; MB LoadOut  DOWN
LB1052 E0_10.08 BOOL  ; MB LoadOut  DOWN CONF
LB1053 E0_10.09 BOOL  ; MB LoadOut Unit DOWN
LB1054 E0_10.10 BOOL  ; MB LoadOut Unit DOWN CONF
LB1055 E0_10.11 BOOL  ; MAGNETIZE 2 START
LB1056 E0_10.12 BOOL  ; MAGNETIZE 2 CONF
LB1057 E0_10.13 BOOL  ; MB LoadOut  UP
LB1058 E0_10.14 BOOL  ; MB LoadOut UP CONF
LB1059 E0_10.15 BOOL  ; MB LoadOut UNIT UP
LB106 E0_11.00 BOOL  ; Take in Slide
LB1060 E0_11.01 BOOL  ; MB LoadOut UNIT UP CONF
LB1061 E0_11.02 BOOL  ; M&B LOAD UNIT SLIDE ADV.
LB1062 E0_11.03 BOOL  ; M&B LOAD UNIT SLIDE ADV. CONF
LB1063 E0_11.04 BOOL  ; MB LoadOut  DOWN
LB1064 E0_11.05 BOOL  ; MB LoadOut DOWN CONF
LB1065 E0_11.06 BOOL  ; MB LoadOut Unit  DOWN
LB1066 E0_11.07 BOOL  ; MB LoadOut UNIT DOWN CONF
LB1067 E0_11.08 BOOL  ; M&B LOAD OUT DEMAGNETIZE START
LB1068 E0_11.09 BOOL  ; M&B LOAD OUT DEMAGNETIZW START CONF
LB1069 E0_11.10 BOOL  ; MB LoadOut  UP
LB1070 E0_11.11 BOOL  ; MB LoadOut  UP CONF
LB1071 E0_11.12 BOOL  ; MB LoadOut  Unit UP
LB1072 E0_11.13 BOOL  ; MB LoadOut UNIT UP CONF
LB1073 E0_11.14 BOOL  ; M&B LOAD UNIT SLIDE RET.
LB1074 E0_11.15 BOOL  ; M&B LOAD UNIT SLIDE RET. CONF
LB1196 E0_12.00 BOOL  ; P11  Case1 Pre-End
LB1197 E0_12.01 BOOL  ; P11  Case2 Pre-End
LB1198 E0_12.02 BOOL  ; P11 Case3 Pre-End
LB1199 E0_12.03 BOOL  ; P11 AutoCycleEnd
LB340 E0_12.04 BOOL  ; IND 1 CYCLE
LB4543 E0_47.14 BOOL  ; dummy on magnet fall memory
LT1012 T3013 TIMER
LT1021 T3014 TIMER
LT1062 T3015 TIMER
LT1068 T3016 TIMER
LT32413 T3042 TIMER
LT420 T3027 TIMER
LT432 T3030 TIMER
LT433 T3041 TIMER
LT5400 T3037 TIMER
LT765 T3023 TIMER
LT941 T3017 TIMER
Mem_Start E0_12.05 BOOL
PH_3304_15_OFF E0_46.03 BOOL
SLIDE_ADV_RTN E0_46.07 BOOL
dbg231 E0_47.09 BOOL
dbug E0_12.06 BOOL
dbug_disch E0_12.07 BOOL
fffe E0_47.08 BOOL
lt433 E0_46.05 BOOL
tes_mg1_off E0_12.08 BOOL
tes_mg1_on E0_12.09 BOOL
tes_mg2_off E0_12.10 BOOL
tes_mg2_on E0_12.11 BOOL
tst_high E0_12.12 BOOL

### Section HMI_Output

